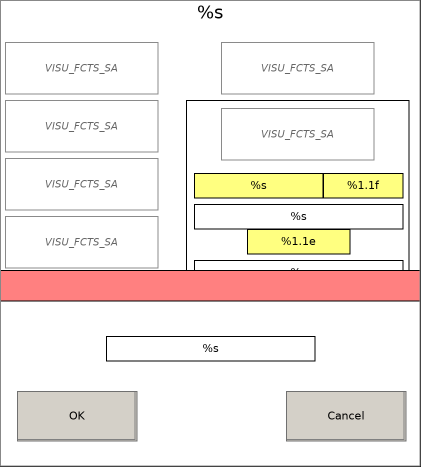
VISUALIZATION SA_POMP_1E_PCR_PPM_ASS  // 421x467
VAR_IN_OUT
	m_Input_PRG:			BLOCK_PRG_POMPAGE;
	m_Input_Jauge:			BLOCK_BCG450_ETHERCAT;
	m_Input_Process:		BLOCK_CDG_ETHERCAT;
	m_Input_Vanne:			BLOCK_VVAT_650_ETHERCAT;
	m_Input_Machine:		BLOCK_MODE_MARCHE_V2_0;
END_VAR
    Rectangle (0,0 421x467), "%s", text list: 'TextList_Navigation', text index: 6
    Frame (5,42 153x52)
        shows VISU_FCTS_SA(m_Input_ID_XML := 1, m_Input_UserRight := PRG_USER.ACTU_USER.FONCTION_SA, m_Input_Operation := m_Input_PRG.POMPAGE.OP_Marche_Pompes)
    Rectangle (74,391 63x25), "%s", text variable: m_Input_Jauge.MNEMO
    Rectangle (144,389 192x29), "%1.2e mbar", text variable: m_Input_Jauge.STATE_Pression
    Rectangle (74,425 63x25), "%s", text variable: m_Input_Process.MNEMO
    Rectangle (144,423 192x29), "%1.2e mbar", text variable: m_Input_Process.STATE_Pression
    Frame (5,100 153x52)
        shows VISU_FCTS_SA(m_Input_ID_XML := 0, m_Input_UserRight := PRG_USER.ACTU_USER.FONCTION_SA, m_Input_Operation := m_Input_PRG.POMPAGE.OP_Pompage_Sec)
    Frame (5,216 153x52)
        shows VISU_FCTS_SA(m_Input_ID_XML := 3, m_Input_UserRight := PRG_USER.ACTU_USER.FONCTION_SA, m_Input_Operation := m_Input_PRG.POMPAGE.OP_Isolement)
    Frame (4,334 153x52)
        shows VISU_FCTS_SA(m_Input_ID_XML := 17, m_Input_UserRight := FALSE, m_Input_Operation := m_Input_PRG.POMPAGE.OP_Regen)
    Frame (5,274 153x52)
        shows VISU_FCTS_SA(m_Input_ID_XML := 4, m_Input_UserRight := PRG_USER.ACTU_USER.FONCTION_SA, m_Input_Operation := m_Input_PRG.POMPAGE.OP_Ventilation)
    Rectangle (186,100 223x274)
    Frame (221,108 153x52)
        shows VISU_FCTS_SA(m_Input_ID_XML := 11, m_Input_UserRight := PRG_USER.ACTU_USER.FONCTION_SA, m_Input_Operation := m_Input_PRG.POMPAGE.OP_Pompage_Proc)
    RoundedRectangle (194,173 129x25), "%s", invisible if: NOT m_Input_Vanne.PRM_Mode, input disabled if: NOT (PRG_USER.ACTU_USER.FONCTION_SA AND NOT m_Input_MACHINE.STATE_Prod) OR m_Input_MACHINE.STATE_Prod, text list: 'TextList_VVAT_650_ETHERCAT', text index: 8
        OnMouseClick: toggle m_Input_Vanne.PRM_Mode
    RoundedRectangle (194,173 129x25), "%s", invisible if: m_Input_Vanne.PRM_Mode, input disabled if: NOT (PRG_USER.ACTU_USER.FONCTION_SA AND NOT m_Input_MACHINE.STATE_Prod) OR m_Input_MACHINE.STATE_Prod, text list: 'TextList_VVAT_650_ETHERCAT', text index: 7
        OnMouseClick: toggle m_Input_Vanne.PRM_Mode
    RoundedRectangle (194,204 209x25), "%s", invisible if: NOT m_Input_Vanne.PRM_Mode, text list: 'TextList_VVAT_650_ETHERCAT', text index: 4
    RoundedRectangle (194,260 209x25), "%s", invisible if: NOT m_Input_Vanne.PRM_Mode, text list: 'TextList_VVAT_650_ETHERCAT', text index: 5
    RoundedRectangle (194,316 209x25), "%s", invisible if: NOT m_Input_Vanne.PRM_Mode, text list: 'TextList_VVAT_650_ETHERCAT', text index: 6
    RoundedRectangle (247,341 103x25), "%s", text variable: m_Input_Vanne.PRM_Tim_W_Pr, invisible if: NOT m_Input_Vanne.PRM_Mode, input disabled if: NOT (PRG_USER.ACTU_USER.FONCTION_SA AND NOT m_Input_MACHINE.STATE_Prod) OR m_Input_MACHINE.STATE_Prod
        OnMouseClick: write the text variable via InputWithLimits
    RoundedRectangle (247,285 103x25), "%1.1e", text variable: m_Input_Vanne.PRM_W_Pr_HI, invisible if: NOT m_Input_Vanne.PRM_Mode, input disabled if: NOT (PRG_USER.ACTU_USER.FONCTION_SA AND NOT m_Input_MACHINE.STATE_Prod) OR m_Input_MACHINE.STATE_Prod
        OnMouseClick: write the text variable via InputWithLimits, min 0, max 1000
    RoundedRectangle (247,229 103x25), "%1.1e", text variable: m_Input_Vanne.PRM_W_Pr_LO, invisible if: NOT m_Input_Vanne.PRM_Mode, input disabled if: NOT (PRG_USER.ACTU_USER.FONCTION_SA AND NOT m_Input_MACHINE.STATE_Prod) OR m_Input_MACHINE.STATE_Prod
        OnMouseClick: write the text variable via InputWithLimits, min 0, max 1000
    RoundedRectangle (323,173 80x25), "%1.1e", text variable: m_Input_Vanne.PRM_Pression, invisible if: NOT m_Input_Vanne.PRM_Mode, input disabled if: NOT (PRG_USER.ACTU_USER.FONCTION_SA AND NOT m_Input_MACHINE.STATE_Prod) OR m_Input_MACHINE.STATE_Prod
        OnMouseClick: write the text variable via InputWithLimits, min 0, max 1000
    RoundedRectangle (323,173 80x25), "%1.1f", text variable: m_Input_Vanne.PRM_Position, invisible if: m_Input_Vanne.PRM_Mode, input disabled if: NOT (PRG_USER.ACTU_USER.FONCTION_SA AND NOT m_Input_MACHINE.STATE_Prod) OR m_Input_MACHINE.STATE_Prod
        OnMouseClick: write the text variable via InputWithLimits, min 0, max 100
    Frame (221,42 153x52)
        shows VISU_FCTS_SA(m_Input_ID_XML := 2, m_Input_UserRight := PRG_USER.ACTU_USER.FONCTION_SA, m_Input_Operation := m_Input_PRG.POMPAGE.OP_Arret_Pompes)
    Frame (5,158 153x52)
        shows VISU_FCTS_SA(m_Input_ID_XML := 28, m_Input_UserRight := PRG_USER.ACTU_USER.FONCTION_SA, m_Input_Operation := m_Input_PRG.POMPAGE.OP_Pompage_Prim)
    Button (4,334 120x50), "%s", input disabled if: NOT m_Input_PRG.POMPAGE.OP_Regen.Autor_IHM OR NOT (PRG_USER.ACTU_USER.FONCTION_SA AND NOT m_Input_Machine.STATE_PROD), text list: 'TextList_SA_Operations', text index: 17
        OnMouseClick: execute { Global_Variables.SHOW_CONFIRM_REGEN:=(TRUE); }
    Group (0,270 421x197), invisible if: NOT Global_Variables.SHOW_CONFIRM_REGEN
        Rectangle (0,0 421x197)
        Button (17,121 120x50), "OK", input disabled if: NOT m_Input_PRG.POMPAGE.OP_Regen.Autor_IHM OR NOT (PRG_USER.ACTU_USER.FONCTION_SA AND NOT m_Input_Machine.STATE_PROD)
            OnMouseClick: execute { m_Input_PRG.POMPAGE.OP_Regen.ON_IHM:=(TRUE); Global_Variables.SHOW_CONFIRM_REGEN:=(FALSE); }
        Button (286,121 120x50), "Cancel"
            OnMouseClick: execute { Global_Variables.SHOW_CONFIRM_REGEN:=(FALSE); }
        Rectangle (0,0 421x31)
        RoundedRectangle (106,66 209x25), "%s", text list: 'TextList_Pompage', text index: 1
END_VISUALIZATION

(* stored: Version 1.1.0.1, ProductVersion 3.1.4024.10
   Visu SA_POMP_1E_PCR_PPM_ASS: Id {caf8e4c6-7a6d-457f-941c-a4162e473ff9} *)
